FUNCTION_BLOCK PMLStateMachine IMPLEMENTS IPmlStateMachine
VAR_INPUT
END_VAR
VAR_OUTPUT
END_VAR
VAR
	_pmlStateMachine : Tc3_PackML_V2.PML_StateMachine;
	_pmlModeMachine : Tc3_PackML_V2.PML_UnitModeManager;
	_subUnits : ARRAY[0..9] OF IPmlStateMachine;
	subUnitArray : ARRAY[0..9] OF ST_PMLSubUnitInfo;
	_SubUnitReference: ST_PMLSubUnitInfoRef;
	i: DINT;
END_VAR

IF _SubUnitReference.NoOfSubUnits <> 0 THEN
	FOR i := 0 TO 9 DO
		IF _subUnits[i] <> 0 THEN
			subUnitArray[i].eState := _subUnits[i].GetCurrentState();
			subUnitArray[i].Active := True;
		END_IF
	END_FOR
	_SubUnitReference.pArray := ADR(subUnitArray);
	_SubUnitReference.ArraySize := SIZEOF(subUnitArray);
END_IF

_pmlStateMachine(eMode := _pmlModeMachine.eModeStatus, stSubUnitInfoRef := _SubUnitReference);
_pmlModeMachine(eState := _pmlStateMachine.eState);

METHOD PUBLIC GetCurrentMode : E_PmlProtectedUnitMode
VAR_INPUT
END_VAR
GetCurrentMode := _pmlModeMachine.eModeStatus;
END_METHOD

METHOD PUBLIC GetCurrentState : E_PMLState
VAR_INPUT
END_VAR
GetCurrentState := _pmlStateMachine.eState;
END_METHOD

METHOD PUBLIC PmlModeCommand : Bool
VAR_INPUT
	Mode : E_PMLProtectedUnitMode;
END_VAR
_pmlModeMachine.eModeCommand := Mode;
END_METHOD

METHOD PUBLIC PmlStateCommand : BOOL
VAR_INPUT
	Command : E_PMLCommand;
END_VAR
_pmlStateMachine.eCommand := Command;
END_METHOD

METHOD PUBLIC RegisterSubUnit : IPmlStateMachine
VAR_INPUT
	SubUnit : IPmlStateMachine;
END_VAR
FOR i := 0 TO 9 DO
	IF _subUnits[i] = 0 THEN
		_subUnits[i] := SubUnit;
		_SubUnitReference.NoOfSubUnits := i + 1;
		EXIT;
	END_IF
END_FOR
END_METHOD

METHOD PUBLIC SetStateComplete : BOOL
VAR_INPUT
END_VAR
_pmlStateMachine.M_StateComplete();
END_METHOD

END_FUNCTION_BLOCK

(* stored: Version 1.1.0.1, ProductVersion 3.1.4024.12
   POU PMLStateMachine: Id {4f8e95fc-32ef-4a74-83fd-0b9512d379fe}, SpecialFunc None
   Method GetCurrentMode: Id {7b17abef-31a4-4387-93cc-006ed2905222}
   Method GetCurrentState: Id {8479c0e8-3207-48b3-b8df-7152ee5b03db}
   Method PmlModeCommand: Id {dc0b200c-2d34-426a-8bf0-20694991bfff}
   Method PmlStateCommand: Id {01ffd23f-e5b1-49e5-90a0-bce9c38c4bb2}
   Method RegisterSubUnit: Id {2bdb4e5c-f6a3-4bbf-b17b-def1b8843c9f}
   Method SetStateComplete: Id {54ff6d39-a4a9-48c3-861d-183e6664d388} *)
